# B&R Automation Studio project LAB3FINAL
Automation Studio 

## Configuration Real

### Task classes (Cpu.sw)
```
Cyclic#1 (cycle 2000 us, tolerance 0 us):
  ncsdcctrl <- ncsdcctrl.prg
  SDCAxisCtr <- SDCAxisCtr.prg
DataObjects: Arnc0sys
NcDataObjects: AxisInit <- AxisInit.dob, gAxis03a <- gAxis03obj.gAxis03a.dob, gAxis03i <- gAxis03obj.gAxis03i.dob, AxisApt <- AxisApt.dob, gmcipvar <- GmcIpUserConfig.gmcipvar.dob, gmcipfun <- GmcIpUserConfig.gmcipfun.dob, gmcipfub <- GmcIpUserConfig.gmcipfub.dob, gmcipubr <- GmcIpUserConfig.gmcipubr.dob, gmcipusm <- GmcIpUserConfig.gmcipusm.dob, gmcipui <- GmcIpUserConfig.gmcipui.dob, gmcipus <- GmcIpUserConfig.gmcipus.dob, gmcipuc <- GmcIpUserConfig.gmcipuc.dob, gmcipsys <- GmcIpConfig.gmcipsys.dob, gmciplbr <- GmcIpConfig.gmciplbr.dob, gmcipcbr <- GmcIpConfig.gmcipcbr.dob, gmciplsm <- GmcIpConfig.gmciplsm.dob, gmcipcsm <- GmcIpConfig.gmcipcsm.dob, gmcipcfg <- GmcIpConfig.gmcipcfg.dob, gmcipiec <- GmcIpConfig.gmcipiec.dob, gmciplog <- GmcIpConfig.gmciplog.dob, gmcipesm <- GmcIpConfig.gmcipesm.dob, gmcipmxd <- GmcIpConfig.gmcipmxd.dob, gmcipmx <- GmcIpConfig.gmcipmx.dob, CncInit <- CncInit.dob, CncProg <- CncProg.dob
Binaries: TCData, Acp10map1, acp10cfg, Acp10map, arconfig, User, Role, sysconf, iomap, asfw, ashwd, arnc0cfg, Arnc0map
Libraries: Acp10sdc, Library, Acp10man, Acp10_MC, sys_lib, brsystem, asstring, powerlnk, asieccon, AsMath, Arnc0man, DataObj, AsArLog, FileIO, AsArProf, AsMem, Runtime, astime, Acp10par, NcGlobal, asiotime
```

### Hardware
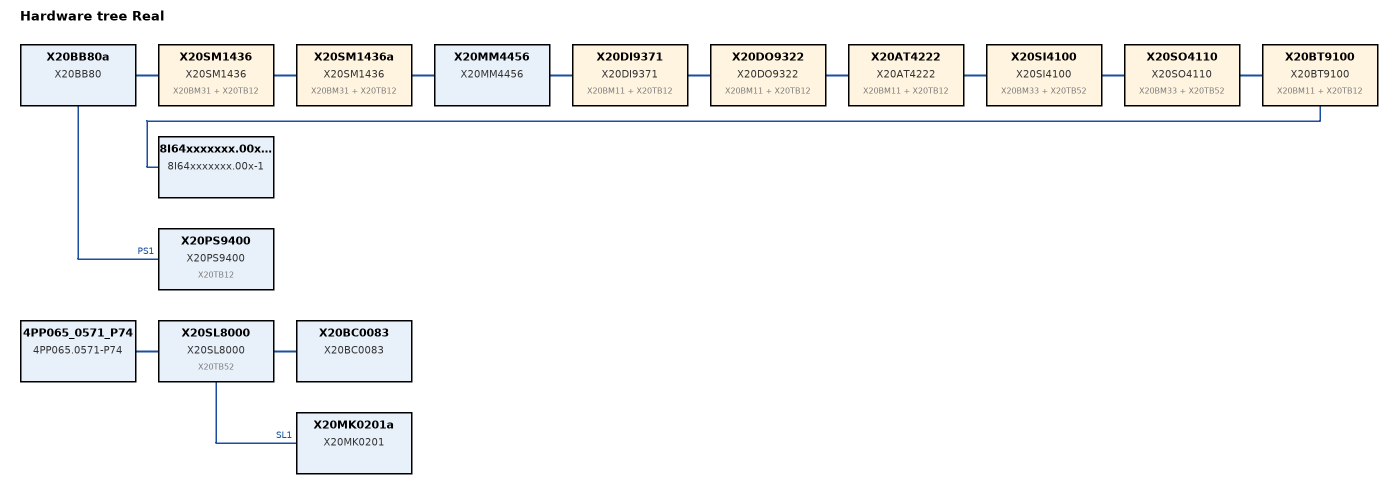
```
4PP065_0571_P74 : 4PP065.0571-P74 v1.1.2.0
  Connector IF4:
    EplInterfaceRedundant = 0
    EplEthInterfaceRedundant = 0
  Connector IF5:
    ActivateDevice = 1
    Mode = Manual
    InternetAddress = 10.0.1.14
    SubnetMask = 255.255.255.0
  ConfigurationID = labBR
  TimerDeviceType = EPLX2X
  TimerDevice = 4PP065_0571_P74.IF4
  TaskClassIdleTime = 2000
  Cyclic1Duration = 2000
  Cyclic1Tolerance = 0
  Cyclic1Output = 1
  Cyclic3Tolerance = 0
  VcObjectName = Visu
8I64xxxxxxx.00x-1 : 8I64xxxxxxx.00x-1 v2.1.2.0  [X2X1 -> X20BT9100.X2X1 [Cable Type=X2XCable, Length=10, Version=1.0.0.2]]
  BothEndSwitchesAreNormallyOpen_r1 = on
  QuickStopIsNormallyOpen_r1 = on
X20AT4222 : X20AT4222 v1.2.3.0  [SS1 -> X20TB12f.SS; SL -> X20BM11c.SL1]
X20BB80a : X20BB80 v1.0.2.0
X20BC0083 : X20BC0083 v2.9.0.0  [PLK1 -> X20SL8000.PLK2 (NodeNumber=2) [Cable Type=PowerlinkCable, Length=10, Version=1.0.0.2]; SL -> X20BB80a.SL1]
X20BM11a : X20BM11 v1.0.0.1  [X2X1 -> X20MM4456.X2X2]
X20BM11b : X20BM11 v1.0.0.1  [X2X1 -> X20BM11a.X2X2]
X20BM11c : X20BM11 v1.0.0.1  [X2X1 -> X20BM11b.X2X2]
X20BM11d : X20BM11 v1.0.0.1  [X2X1 -> X20BM33b.X2X2]
X20BM31a : X20BM31 v1.0.0.1  [X2X1 -> X20BB80a.IF1]
X20BM31b : X20BM31 v1.0.0.1  [X2X1 -> X20BM31a.X2X2]
X20BM33a : X20BM33 v1.0.0.4  [X2X1 -> X20BM11c.X2X2]
X20BM33b : X20BM33 v1.0.0.4  [X2X1 -> X20BM33a.X2X2]
X20BT9100 : X20BT9100 v1.0.3.0  [SS1 -> X20TB12g.SS; SL -> X20BM11d.SL1]
X20DI9371 : X20DI9371 v1.0.2.0  [SS1 -> X20TB12d.SS; SL -> X20BM11a.SL1]
X20DO9322 : X20DO9322 v1.0.3.0  [SS1 -> X20TB12e.SS; SL -> X20BM11b.SL1]
X20MK0201a : X20MK0201 v1.0.0.0  [SL -> X20SL8000.SL1]
X20MM4456 : X20MM4456 v1.4.0.0  [X2X1 -> X20BM31b.X2X2]
X20PS9400 : X20PS9400 v1.0.2.4  [SS1 -> X20TB12b.SS; PS -> X20BB80a.PS1]
X20SI4100 : X20SI4100 v1.10.1.1  [SS1 -> X20TB52b.SS; SL -> X20BM33a.SL1]
X20SL8000 : X20SL8000 v1.6.5.1  [PLK1 -> 4PP065_0571_P74.IF4 (NodeNumber=1) [Cable Type=PowerlinkCable, Length=10, Version=1.0.0.2]; PLK2 -> X20BC0083.PLK1 (NodeNumber=1) [Cable Type=PowerlinkCable, Length=10, Version=1.0.0.2]; SS1 -> X20TB52a.SS]
  SafeProject = SafeLOGIC-1
X20SM1436 : X20SM1436 v1.4.2.1  [SS1 -> X20TB12a.SS; SL -> X20BM31a.SL1]
X20SM1436a : X20SM1436 v1.4.2.1  [SS1 -> X20TB12c.SS; SL -> X20BM31b.SL1]
X20SO4110 : X20SO4110 v1.10.1.1  [SS1 -> X20TB52c.SS; SL -> X20BM33b.SL1]
  SafeLogicID = 2
  SafeModuleID = 3
X20TB12a : X20TB12 v1.0.0.0
X20TB12b : X20TB12 v1.0.0.0
X20TB12c : X20TB12 v1.0.0.0
X20TB12d : X20TB12 v1.0.0.0
X20TB12e : X20TB12 v1.0.0.0
X20TB12f : X20TB12 v1.0.0.0
X20TB12g : X20TB12 v1.0.0.0
X20TB52a : X20TB52 v1.0.0.1
X20TB52b : X20TB52 v1.0.0.1
X20TB52c : X20TB52 v1.0.0.1
```

### IoMap.iom - 4PP065_0571_P74/IoMap.iom
```iecst
VAR_CONFIG
	Cyclic#1.gAxis03_DrvIf.iLifeCnt AT %IB."8I64xxxxxxx.00x-1".SDC_LifeCnt;
	Cyclic#1.gAxis03_DrvIf.iDrvOK AT %IX."8I64xxxxxxx.00x-1".ETAD_Input_Bool_02;
	Cyclic#1.gAxis03_DrvIf.oSetTime AT %QW."8I64xxxxxxx.00x-1".SDC_SetTime;
	Cyclic#1.gAxis03_DrvIf.oSetPos AT %QW."8I64xxxxxxx.00x-1".LFRD_Output;
	Cyclic#1.gAxis03_DiDoIf.iLifeCntDriveReady AT %IB."8I64xxxxxxx.00x-1".SDC_LifeCnt;
	Cyclic#1.gAxis03_DiDoIf.iLifeCntDriveEnable AT %IB."8I64xxxxxxx.00x-1".SDC_LifeCnt;
	Cyclic#1.gAxis03_DiDoIf.oDriveEnable AT %QX."8I64xxxxxxx.00x-1".CMDD_Output_Bool_00;
	Cyclic#1.gAxis03_ModuleOk AT %QX."8I64xxxxxxx.00x-1".CMDD_Output_Bool_01;
	Cyclic#1.gAxis03_ModuleOk AT %QX."8I64xxxxxxx.00x-1".CMDD_Output_Bool_02;
	Cyclic#1.gAxis03_ModuleOk AT %IX."8I64xxxxxxx.00x-1".ModuleOk;
	Cyclic#1.gAxis03_DiDoIf.oDriveEnable AT %QX."8I64xxxxxxx.00x-1".CMDD_Output_Bool_03;
	Cyclic#1.gAxis03_DiDoIf.iDriveReady AT %IX."8I64xxxxxxx.00x-1".ETAD_Input_Bool_02;
	::SDCAxisCtr:pwm_period AT %QW."X20MM4456".PeriodDurationPWM;
	::SDCAxisCtr:axis_X.pwm_value AT %QW."X20MM4456".PulseWidthCurrentPWM01;
	::SDCAxisCtr:axis_X.reset_error AT %QX."X20MM4456".ClearError01;
	::SDCAxisCtr:axis_X.reset_counter AT %QX."X20MM4456".ResetCounter01;
	::SDCAxisCtr:axis_X.counter AT %IW."X20MM4456".Counter01;
	::SDCAxisCtr:axis_X.endswitch_a_reached AT %IX."X20MM4456".StatusInput03; (*Logical condition input 01=Motor 01:A*)
	::SDCAxisCtr:axis_X.endswitch_b_reached AT %IX."X20MM4456".StatusInput04; (*Logical condition input 02=Motor 01:B*)
	::SDCAxisCtr:coil_powered AT %IX."X20DI9371".DigitalInput01;
END_VAR
```

### Acp10map1.ncm - 4PP065_0571_P74/Motion/Acp10map1.ncm
```
NcMapping (NcSwId=ACP10, DisabledNodesAreHidden=False)
  NcObject AxisX (ModuleAddress=SDC_IF1.ST2, InterfaceType=SDC, Type=ncAXIS, Channel=1, AcoposSimulation=Off, InitParameter=AxisInit, AcoposParameter=AxisApt, AdditionalData=CNC_Enabled="1" , Disabled=FALSE, ModuleDisabled=FALSE)
  NcObject AxisY (ModuleAddress=SDC_IF1.ST3, InterfaceType=SDC, Type=ncAXIS, Channel=1, AcoposSimulation=Off, InitParameter=AxisInit, AcoposParameter=AxisApt, AdditionalData=CNC_Enabled="1" , Disabled=FALSE)
  NcObject AxisZ (ModuleAddress=SDC_IF1.ST4, InterfaceType=SDC, Type=ncAXIS, Channel=1, AcoposSimulation=Off, InitParameter=AxisInit, AcoposParameter=AxisApt, AdditionalData=CNC_Enabled="1" , Disabled=FALSE)
```


## Logical view

Binary libraries used (declarations not repeated): Runtime, Operator, AsIecCon, astime, Acp10sdc, Acp10man, Acp10par, NcGlobal, asstring, AsIOTime, Acp10_MC, brsystem, sys_lib, Acp10sim, AsMath, Arnc0man, DataObj, AsArLog, FileIO, AsArProf, AsMem

### Global.var - Global variables
```iecst
VAR
	AxisX : ACP10AXIS_typ := (0);
	AxisX_EncIf : SdcEncIf16_typ := (0);
	AxisX_DrvIf : SdcDrvIf16_typ := (0);
	AxisX_DiDoIf : SdcDiDoIf_typ := (0);
	AxisX_HW : SdcHwCfg_typ := (0);
	gAxisTest : ACP10AXIS_typ := (0);
	gAxisTest_HW : SdcHwCfg_typ := (0);
	gAxisTest_DrvIf : SdcDrvIf16_typ := (0);
	gAxisTest_DiDoIf : SdcDiDoIf_typ := (0);
	gAxisTest_ModuleOk : BOOL := 0;
	gAxis03 : ACP10AXIS_typ := (0);
	gAxis03_HW : SdcHwCfg_typ := (0);
	gAxis03_DrvIf : SdcDrvIf16_typ := (0);
	gAxis03_DiDoIf : SdcDiDoIf_typ := (0);
	gAxis03_ModuleOk : BOOL := 0;
	CNCsys : ARNC0CNC_typ;
END_VAR
```

### Package Logical/Libraries - Global libraries

### Library Logical/Libraries/Library (ANSIC)

#### FB_Axis.c
```c
#include <bur/plctypes.h>
#ifdef __cplusplus
	extern "C"
	{
#endif
	#include "Library.h"
#ifdef __cplusplus
	};
#endif
/* TODO: Add your comment here */
void FB_Axis(struct FB_Axis* inst)
{
	/*
	if (inst->pwm_percentage > 100)
	{
		inst->pwm_percentage = 100;
	}
	if (inst->pwm_percentage < -100)
	{
		inst->pwm_percentage = -100;
	}
	REAL raw_percentage = (REAL) inst->pwm_percentage / 100.0 * 32767.0;
	inst->pwm_value = (INT) raw_percentage;
	*/
	inst->speed = inst->counter - inst->last_counter;
	inst->speed = (inst->speed * 3000 / 24.0) / 0.002;
	inst->last_counter = inst->counter;
}
```

#### FB_Motor.c
```c
#include <bur/plctypes.h>
#ifdef __cplusplus
	extern "C"
	{
#endif
	#include "Library.h"
#ifdef __cplusplus
	};
#endif
/* TODO: Add your comment here */
void FB_Motor(struct FB_Motor* inst)
{
	REAL a = inst->in / inst->k_e - inst->out_w;
	REAL b = a / inst->T_m;
	inst->integrator.dt = inst->dt;
	inst->integrator_phi.dt = inst->dt;
	inst->integrator.in = b;
	FB_Integrator(&inst->integrator);
	inst->out_w = inst->integrator.out;
	inst->integrator_phi.in = inst->out_w;
	FB_Integrator(&inst->integrator_phi);
	inst->out_phi = inst->integrator_phi.out;
}
```

### Package Logical/gAxis03obj - gAxis03obj

### gAxis03i.ax
```
InitParameter (Version=3.13.1, NcSwId=Acp10)
  ACP10AXIS_typ:
    dig_in:
      level:
        reference = ncACTIV_HI
        pos_hw_end = ncACTIV_HI
        neg_hw_end = ncACTIV_HI
        trigger1 = ncACTIV_HI
        trigger2 = ncACTIV_HI
    encoder_if:
      parameter:
        count_dir = ncSTANDARD
        scaling:
          load:
            units = 1000
            rev_motor = 1
    limit:
      parameter:
        v_pos = 10000
        v_neg = 10000
        a1_pos = 50000
        a2_pos = 50000
        a1_neg = 50000
        a2_neg = 50000
        t_jolt = 0
        t_in_pos = 0
        pos_sw_end = 2000000000
        neg_sw_end = -2000000000
        ds_warning = 500
        ds_stop = 1000
        a_stop = 1.0e30
        dv_stop = 0
        dv_stop_mode = ncOFF
    controller:
      mode = ncPOSITION
      position:
        kv = 50
        tn = 0
        t_predict = 0.01
        t_total = 0.01
        p_max = 1.0e30
        i_max = 0
      speed:
        kv = 2.0
        tn = 0
        t_filter = 0.0
        isq_filter1:
          type = ncOFF
          a0 = 0.0
          a1 = 0.0
          b0 = 0.0
          b1 = 0.0
          b2 = 0.0
          c0_par_id = 0
          c1_par_id = 0
        isq_filter2:
          type = ncOFF
          a0 = 0.0
          a1 = 0.0
          b0 = 0.0
          b1 = 0.0
          b2 = 0.0
          c0_par_id = 0
          c1_par_id = 0
        isq_filter3:
          type = ncOFF
          a0 = 0.0
          a1 = 0.0
          b0 = 0.0
          b1 = 0.0
          b2 = 0.0
          c0_par_id = 0
          c1_par_id = 0
      uf:
        type = ncLINEAR
        auto_config = ncMOTOR_PAR
        u0 = 0
        un = 0
        fn = 50.0
        k_f_slip = 0
      ff:
        torque_load = 0.0
        torque_pos = 0.0
        torque_neg = 0.0
        kv_torque = 0.0
        inertia = 0.0
        t_filter_a = 0.0
    move:
      stop:
        parameter[0]:
          decel_ramp = ncA_LIMIT
          controller = ncON
        parameter[1]:
          decel_ramp = ncA_LIMIT
          controller = ncON
        parameter[2]:
          decel_ramp = ncA_LIMIT
          controller = ncON
        parameter[3]:
          decel_ramp = ncA_LIMIT
          controller = ncON
        quickstop:
          decel_ramp = ncA_LIMIT
        drive_error:
          decel_ramp = ncA_LIMIT
      homing:
        parameter:
          s = 0
          v_switch = 5000
          v_trigger = 500
          a = 50000
          mode = ncDIRECT
          edge_sw = ncPOSITIVE
          start_dir = ncPOSITIVE
          trigg_dir = ncPOSITIVE
          ref_pulse = ncOFF
          fix_dir = ncOFF
          tr_s_block = 0
          torque_lim = 0
          ds_block = 0
          ds_stop = 0
      basis:
        parameter:
          v_pos = 5000
          v_neg = 5000
          a1_pos = 50000
          a2_pos = 50000
          a1_neg = 50000
          a2_neg = 50000
    message:
      text:
        parameter:
          format = ncBREAK
          columns = 80
          data_modul = acp10etxen
```

- Data object Logical/GmcIpConfig/gmcipsys (Cnc, version 3.13.0) (no source held here)

### Data object Logical/GmcIpConfig/gmciplbr (Cnc)

#### gmciplbr.cnc
```
Root (LangModule=ailgcode, Version=1.0)
  BuiltInProcs:
    cancel = beginpathsynch
        StopCyclicGroups(:${*}:);
      endpathsynch (MinArgs=1, MaxArgs=*)
  BuiltInFns (PatternSuffix=:\[)
    ABS = Abs(:$[1]:) (NumArgs=1, Inline=Yes)
    SQR = ($[1] * $[1]) (NumArgs=1)
    ACOS = ACos(:$[1]:) (NumArgs=1, Inline=Yes)
    ASIN = ASin(:$[1]:) (NumArgs=1, Inline=Yes)
    ATAN = ATan(:$[1]:) (NumArgs=1, Inline=Yes)
    COS = Cos(:$[1]:) (NumArgs=1, Inline=Yes)
    DEXP = DExp(:$[1]:) (NumArgs=1, Inline=Yes)
    EXP = Exp(:$[1]:) (NumArgs=1, Inline=Yes)
    FIX = Fix(:$[1]:) (NumArgs=1, Inline=Yes)
    FRACT = Fract(:$[1]:) (NumArgs=1, Inline=Yes)
    FUP = Fup(:$[1]:) (NumArgs=1, Inline=Yes)
    INV = ~($[1]) (NumArgs=1, Inline=Yes)
    LN = Ln(:$[1]:) (NumArgs=1, Inline=Yes)
    LOG = Log(:$[1]:) (NumArgs=1, Inline=Yes)
    ROUND = ToInt(:$[1]:) (NumArgs=1, Inline=Yes)
    SIN = Sin(:$[1]:) (NumArgs=1, Inline=Yes)
    SQRT = Sqrt(:$[1]:) (NumArgs=1, Inline=Yes)
    TAN = Tan(:$[1]:) (NumArgs=1, Inline=Yes)
    BOOL = ToBool(:$[1]:) (NumArgs=1, Inline=Yes)
    INT = Fix(:$[1]:) (NumArgs=1, Inline=Yes)
    ADR = Adr(:\$[1]:) (NumArgs=1, Inline=Yes)
    SIZEOF = Sizeof(:\$[1]:) (NumArgs=1, Inline=Yes)
    NUM_LOADED_FILES = NumLoadedFiles(::) (NumArgs=0)
    NUM_LOADED_PROG_FILES = NumLoadedProgFiles(::) (NumArgs=0)
    MEM_SIZE_IP_ALL = MemSizeIpInstAll(::) (NumArgs=0)
    MEM_SIZE_IP_LIB = MemSizeIpInst(::) (NumArgs=0)
    MEM_SIZE_SHLIB = MemSizeShLib(::) (NumArgs=0)
    MEM_SIZE_FILE = MemSizeFile(:$[1]:) (MinArgs=0, MaxArgs=1)
    MEM_SIZE_IP_STACK_SPACE = MemStackSpace(::) (NumArgs=0)
  AxesSpec:
    AxisRef = $\s*=\s*AC (Mode=3)
    AxisRef = $\s*=\s*IC (Mode=4)
  PVMacros:
    RDISABLE (ArrayDims=0, Group=500)
      CALL = @#job->sa.keep_alive = 1;
        @#thread.sa_keep_alive = 1; (Inline=Yes)
  Parameters:
    R (IndexType=RParamIndex, ValueType=FLOAT)
      ARG (ref=EXPR, DataType=RParamIndex)
    P (IndexType=RParamIndex, ValueType=FLOAT)
      ARG (ref=EXPR, DataType=RParamIndex)
    EXB (IndexType=EXParamIndex, ValueType=Byte)
      ARG (ref=EXPR, DataType=EXParamIndex)
    EXW (IndexType=EXParamIndex, ValueType=Word)
      ARG (ref=EXPR, DataType=EXParamIndex)
    EXL (IndexType=EXParamIndex, ValueType=Long)
      ARG (ref=EXPR, DataType=EXParamIndex)
    EXF (IndexType=EXFParamIndex, ValueType=FLOAT)
      ARG (ref=EXPR, DataType=EXFParamIndex)
    MW (Synchronous=Yes, IndexType=MParamIndex, ValueType=Word)
      ARG (ref=EXPR, DataType=MParamIndex)
    ML (Synchronous=Yes, IndexType=MParamIndex, ValueType=Long)
      ARG (ref=EXPR, DataType=MParamIndex)
    MF (Synchronous=Yes, IndexType=MParamIndex, ValueType=FLOAT)
      ARG (ref=EXPR, DataType=MParamIndex)
  PrimTypes (PatternSuffix=:[^\[], MapIECTypes=Yes)
  Preprocess:
    PP_RULE_FRAME_I (Search=$FRAME_I, Replace=[1,0,0,0,1,0,0,0,1,0,0,0])
    PP_RULE_FRAME_DEF (IsPattern=Yes, Search=FRAME:[^\w\d], Replace=LREAL{12})
  FubTemplates:
    StdFubTemplate (IsDefault=Yes, Inline=Yes)
      Arg (ref=FUBINST, DataType=FLOAT)
      Arg (ref=FUBERRLEV, DataType=FLOAT)
      Arg (ref=PATHSYNCH, DataType=FLOAT)
      Arg (ref=BLOCKING, DataType=FLOAT)
  SynchActions:
    SABlocks:
      default (IsDefault=Yes)
        cyclic (Inline=Yes)
          Arg (ref=ACTIONS, DataType=STATEMENTS)
          Arg (ref=ID, DataType=FLOAT, DefaultInt=-1, MinCount=0, MaxCount=1)
      whenever:
        cyclic (Inline=Yes)
          Arg (ref=COND, DataType=FLOAT)
          Arg (ref=ACTIONS, DataType=STATEMENTS)
          Arg (ref=ID, DataType=FLOAT, DefaultInt=-1, MinCount=0, MaxCount=1)
      when:
        cyclic (Inline=Yes)
          Arg (ref=COND, DataType=FLOAT)
          Arg (ref=ACTIONS, DataType=STATEMENTS)
          Arg (ref=ID, DataType=FLOAT, DefaultInt=-1, MinCount=0, MaxCount=1)
      every:
        cyclic (Inline=Yes)
          Arg (ref=COND, DataType=FLOAT)
          Arg (ref=ACTIONS, DataType=STATEMENTS)
          Arg (ref=ID, DataType=FLOAT, DefaultInt=-1, MinCount=0, MaxCount=1)
      from:
        cyclic (Inline=Yes)
          Arg (ref=COND, DataType=FLOAT)
          Arg (ref=ACTIONS, DataType=STATEMENTS)
          Arg (ref=ID, DataType=FLOAT, DefaultInt=-1, MinCount=0, MaxCount=1)
    NonModalActivation:
      Start = @#thread.sa_last_keep_alive = 1;
        ActivateCyclicGroup(:-1:);
      Stop = WaitStopCyclicGroups(:(:-1:):);
  ParserData (NestedComments=Yes, DefaultCaseSensitive=No, CommentsSpanLines=No, SubDeclsLocalToFile=Yes, ProgDeclsLocalToFile=Yes, AllowUnprefixedFileCalls=No, LocalVarScopeForMainProg=No, FileScopeVarsVisibleInSub=Yes, MainPrgReturnAtNextMainPrgHdr=Yes, MaxSizePassByValue=1024, AllowVarReadBeforeAssign=No, AllowArrayRefWithoutIndex=Yes, AllowStructMemberAutoDereference=Yes, AllowVariableAutoDereference=Yes, AllowIgnoredExtraSubArgs=Yes, EnableStringCharacterIndexing=Yes, OnMacroRedefinition=Warn, CheckFileTimestampBeforeCalls=Yes)
    TKG_END_OF_LINE = \n (IsPattern=No)
    TKG_LINE_CONTINUE = \ (IsPattern=No, FileXLInvalid=Yes)
    TKG_LINE_BREAK = @@
    TKG_ARITH_BINARY_MODULO = MOD
    TKG_TRUE = TRUE:\W (IsPattern=Yes)
    TKG_FALSE = FALSE:\W (IsPattern=Yes)
    TKG_PAREVAL_MODAL_ID = ID:[\s=] (FileXLInvalid=Yes, IsPattern=Yes)
    TKG_OPEN_COMMENT = (
    TKG_CLOSE_COMMENT = )
    TKG_OPEN_BRACKET = [
    TKG_COMMA = ,
    TKG_CLOSE_BRACKET = ]
    TKG_OPEN_INDEXBRACKET = {
    TKG_CLOSE_INDEXBRACKET = }
    TKG_NUMBER = \d+\.\d+|\d+\.:[^\.] (IsPattern=Yes)
    TKG_INTEGER = \d+ (IsPattern=Yes)
    TKG_FRACTION = \.\d+ (IsPattern=Yes)
    TKG_DOT = \.:\w (IsPattern=Yes, FollowedBy=TKG_STRUCT_MEMBER_REF)
    TKG_STRUCT_MEMBER_REF = \w|\w[\w\d]+ (IsPattern=Yes, Restricted=Yes)
    TKG_NUMBER_EXP = EX:[\s\d\+\-\.] (IsPattern=Yes)
    TKG_MACRO_DEFINE_GLOBAL = define\s+ip_global:\s (IsPattern=Yes, FollowedBy=TKG_MACRO_NAME)
    TKG_MACRO_DEFINE = define\s+local:\s|define:\s (IsPattern=Yes, FollowedBy=TKG_MACRO_NAME)
    TKG_MACRO_UNDEFINE = undefine:\s (IsPattern=Yes, FollowedBy=TKG_MACRO_NAME)
    TKG_MACRO_AS = as:[\s\n] (IsPattern=Yes, FollowedBy=TKG_MACRO_TEXT)
    TKG_MACRO_NAME = [$\w][$\w\d]+ (Restricted=Yes, IsPattern=Yes)
    TKG_MACRO_TEXT = . (Restricted=Yes, IsPattern=Yes)
    TKG_BUILTIN_NUM_FN_NAME
    _TKG_LABEL_DEF1:
      TKG_LABEL_DEF = L[\w\d]+:\:[^\w\d] (IsPattern=Yes, FollowedBy=TKG_LABEL_SUFFIX)
    TKG_SUBPROG_START = %:L (FileXLInvalid=Yes, IsPattern=Yes, FollowedBy=TKG_SUBPROG_NAME)
    TKG_SUBPROG_NAME = L\d+ (IsPattern=Yes, Restricted=Yes)
    TKG_SUBPROG_CALL = L:L\d (IsPattern=Yes, FollowedBy=TKG_SUBPROG_NAME)
    TKG_SUBPROG_PROTO = %D:L (IsPattern=Yes, FollowedBy=TKG_SUBPROG_NAME)
    TKG_SUBCALL_REPEAT_PREFIX = O:[\s\d] (IsPattern=Yes, FollowedBy=TKG_INTEGER)
    TKG_EXTERN = EXTERN:\s (IsPattern=Yes, FollowedBy=TKG_PROG_FILE_NAME)
    TKG_ARG_PASSBYREF = VAR\s (IsPattern=Yes)
    TKG_SET_MODAL_SUB = MCALL:\W (FileXLInvalid=Yes, IsPattern=Yes)
    TKG_PROG_START = %:\d (IsPattern=Yes, FollowedBy=TKG_PROG_NAME)
    TKG_PROG_NAME = \d+ (IsPattern=Yes, Restricted=Yes)
    TKG_PROG_CALL = L:[^L] (IsPattern=Yes, FollowedBy=TKG_PROG_FILE_NAME)
    TKG_PROG_FILE_NAME = [\^#&@']?[\w\d\.\\]+:[^\w\d\.\\\:]|[\^#][\w\d]+\:[\w\d\.\\]+ (IsPattern=Yes, Restricted=Yes)
    TKG_SUPPRESS_SINGLE_STEP = NOHALT
    TKG_NC_BLOCK_PREFIX = N:[\d\s] (IsPattern=Yes)
    TKG_PARAM_PREFIX = R:\d|P:\d|M[WLF]:\d|EX[WLBF]:\d (IsPattern=Yes)
    TKG_SUBRANGE = ..
    TKG_G_CODE_PREFIX = G:[\s\d] (IsPattern=Yes)
    TKG_M_CODE_PREFIX = M:[\s\d\[] (IsPattern=Yes)
    TKG_PAREVAL_DO = do:\s (FileXLInvalid=Yes, IsPattern=Yes)
    TKG_GOTO = $GOTO:\s (FileXLInvalid=Yes, IsPattern=Yes, OptFollowedBy=TKG_GOTO_DEST)
    TKG_GOTO_DEST = \w[\w\d]* (IsPattern=Yes, Restricted=Yes)
    TKG_LOGICAL_BINARY_AND = &&
    TKG_LOGICAL_BINARY_OR = ||
    TKG_LOGICAL_BINARY_XOR = XOR
    TKG_STRING_CONCAT = <<
    TKG_COMP_BINARY_GREATER_THAN_OR_EQ = >=
    TKG_COMP_BINARY_LESS_THAN_OR_EQ = <=
    TKG_COMP_BINARY_EQUAL_TO = ==
    TKG_COMP_BINARY_NOT_EQUAL_TO = !=
    TKG_COMP_BINARY_GREATER_THAN = >
    TKG_COMP_BINARY_LESS_THAN = <
    TKG_ASSIGN_EQ = =
    TKG_LOGICAL_UNARY_NOT = !
    TKG_BITWISE_BINARY_AND = &
    TKG_BITWISE_BINARY_OR = |
    TKG_BITWISE_BINARY_XOR = ^
    TKG_BITWISE_UNARY_COMPLEMENT = ~
    TKG_ARITH_BINARY_PLUS = +
    TKG_ARITH_BINARY_MINUS = -
    TKG_ARITH_BINARY_POWER = **
    TKG_ARITH_BINARY_MULTIPLY = *
    TKG_ARITH_BINARY_DIVIDE = /
    TKG_IF = $IF (FileXLInvalid=Yes)
    TKG_THEN = $THEN (FileXLInvalid=Yes)
    TKG_BLOCK_ELSEIF = $ELSEIF (FileXLInvalid=Yes)
    TKG_BLOCK_ELSE = $ELSE (FileXLInvalid=Yes)
    TKG_BLOCK_ENDIF = $ENDIF (FileXLInvalid=Yes)
    TKG_SWITCH = $SWITCH (FileXLInvalid=Yes)
    TKG_SWITCH_CASE = $CASE (FileXLInvalid=Yes)
    TKG_SWITCH_DEFAULT = $DEFAULT (FileXLInvalid=Yes)
    TKG_ENDSWITCH = $ENDSWITCH (FileXLInvalid=Yes)
    TKG_FOR = $FOR (FileXLInvalid=Yes)
    TKG_ENDFOR = $ENDFOR (FileXLInvalid=Yes)
    TKG_WHILE = $WHILE (FileXLInvalid=Yes)
    TKG_ENDWHILE = $ENDWHILE (FileXLInvalid=Yes)
    TKG_DO = $DO (FileXLInvalid=Yes)
    TKG_ENDDO = $ENDDO (FileXLInvalid=Yes)
    TKG_BREAK = $BREAK (FileXLInvalid=Yes)
    TKG_CONTINUE = $CONTINUE (FileXLInvalid=Yes)
    TKG_PRIM_TYPE (IsPattern=Yes)
    TKG_PV_DECL = def:\s (IsPattern=Yes)
    TKG_PV_UNDECL = ~def:\s (IsPattern=Yes)
    TKG_PV_DECL_REF = \w[\w\d\.\:\*]+|\w (IsPattern=Yes, Restricted=Yes)
    TKG_VARSCOPE_IP_LOCAL = local:[\s\n] (IsPattern=Yes)
    TKG_VARSCOPE_IP_GLOBAL = ip_global:[\s\n] (IsPattern=Yes)
    TKG_VARSCOPE_NC_GLOBAL = nc_global:[\s\n] (IsPattern=Yes)
    TKG_VARSCOPE_PLC_GLOBAL = plc_global:[\s\n] (IsPattern=Yes)
    TKG_VAR_RETAIN = retain:\s (IsPattern=Yes)
    TKG_VARSYNCH_IP = ip_synch:\s (IsPattern=Yes)
    TKG_VARSYNCH_PATH = path_synch:\s (IsPattern=Yes)
    TKG_LABEL_DEF = \w:\:|\w[\w\d]+:\: (IsPattern=Yes, FollowedBy=TKG_LABEL_SUFFIX)
    TKG_LABEL_SUFFIX = : (Restricted=Yes)
    TKG_FUB_DECL = fub:\s (IsPattern=Yes)
    TKG_FUB_ERR_LEV_1 = error_level_1:\s (IsPattern=Yes)
    TKG_FUB_ERR_LEV_2 = error_level_2:\s (IsPattern=Yes)
    TKG_FUB_ERR_LEV_3 = error_level_3:\s (IsPattern=Yes)
    TKG_FUB_ERR_LEV_4 = error_level_4:\s (IsPattern=Yes)
    TKG_FUB_BLOCKING = blocking:\s (IsPattern=Yes)
    TKG_FUB_NON_BLOCKING = non_blocking:\s (IsPattern=Yes)
    TKG_IEC_TYPED_VALUE = #[\w\d]+ (IsPattern=Yes)
    TKG_REFERENCE = ref:[\s\n]|reference:[\s\n] (IsPattern=Yes, FollowedBy=TKG_IEC_TO)
    TKG_IEC_TO = to:[\s\n] (IsPattern=Yes, Restricted=Yes)
    TKG_ACCESS = ACCESS:[\s\n] (IsPattern=Yes)
    TKG_WORD = \w|\w[\w\d\.]+ (IsPattern=Yes)
  StringChars (AsciiStringStart=", UTF16StringStart=W", UTF16StringEnd=")
    EscapeSeq (Search=$N, ReplaceValue=10)
    EscapeSeq (Search=$L, ReplaceValue=10)
    EscapeSeq (Search=$P, ReplaceValue=12)
    EscapeSeq (Search=$R, ReplaceValue=13)
    EscapeSeq (Search=$T, ReplaceValue=9)
    EscapeSeq (Search=$Q, ReplaceStr=")
    EscapeSeq (Search=$', ReplaceStr=')
    EscapeSeq (Search=$", ReplaceStr=")
    EscapeSeq (Search=$[\dA-Fa-f]+, IsPattern=Yes, ReplaceEncodingBase=16)
    EscapeSeq (Search=$$, ReplaceStr=$)
    EscapeSeq (Search=$, ReplaceStr=)
```

- Data object Logical/GmcIpConfig/gmcipcbr (Cnc, version 3.13.0) (no source held here)

### Data object Logical/GmcIpConfig/gmcipcsm (Cnc)

#### gmcipcsm.cnc
```
Root (LangModule=ailgcode, Version=1.0)
  Constants:
    NumAxes = 15 (Type=INT)
  Preprocess:
    PP_RULE_STOPRE (Search=STOPRE, Replace=G172)
    PP_RULE_CIP (Search=CIP:\W, Replace=G102, IsPattern=Yes)
  Types:
    RotationAngleSpecifier (type=ENUM, EnumType=REGEXP, Value6=H)
    RadiusSpecifier (type=ENUM, EnumType=REGEXP, Value1=R\s*=, Value2=CR\s*=)
    InterpolParam (type=ENUM, EnumType=REGEXP, Value0=I, Value1=J, Value2=K, Value100=G161\s*I, Value101=G161\s*J, Value102=G161\s*K, Value200=G162\s*I, Value201=G162\s*J, Value202=G162\s*K, Value0300=I\s*=\s*AC, Value0301=J\s*=\s*AC, Value0302=K\s*=\s*AC, Value0400=I\s*=\s*IC, Value0401=J\s*=\s*IC, Value0402=K\s*=\s*IC)
    CirclePointParam (type=ENUM, EnumType=REGEXP, Value0=I1\s*=, Value1=J1\s*=, Value2=K1\s*=, Value100=G161\s*I1\s*=, Value101=G161\s*J1\s*=, Value102=G161\s*K1\s*=, Value200=G162\s*I1\s*=, Value201=G162\s*J1\s*=, Value202=G162\s*K1\s*=, Value0300=I1\s*=\s*AC, Value0301=J1\s*=\s*AC, Value0302=K1\s*=\s*AC, Value0400=I1\s*=\s*IC, Value0401=J1\s*=\s*IC, Value0402=K1\s*=\s*IC)
    RPYAngleName (type=ENUM, EnumType=REGEXP, Value1=ROLL, Value0=PITCH, Value2=YAW)
    EulerAngleName (type=ENUM, EnumType=REGEXP, Value3=PHI, Value4=THETA, Value5=PSI)
    RotaryVectorName (type=ENUM, EnumType=REGEXP, Value0=P\s*=, Value1=Q\s*=, Value2=R\s*=)
    DwellTime (type=FLOAT)
    RParamIndex (type=INT, MinValue=0, MaxValue=999)
    EXParamIndex (type=INT, MinValue=0, MaxValue=99)
    MParamIndex (type=INT, MinValue=0, MaxValue=99)
    Byte (type=INT, MinValue=0, MaxValue=255)
    Word (type=INT, MinValue=-32768, MaxValue=32767)
    Long (type=INT)
  PVMacros:
    SAVE (ArrayDims=0, Group=500)
      CALL = Info(:id:52101, msg:"Save Modal GCode State NOT SUPPORTED YET":);
  SysVars
  Parameters:
    R (IndexType=RParamIndex, ValueType=FLOAT)
      ARG (ref=EXPR, DataType=RParamIndex)
    QUOTED (QuotedName=$R, Synchronous=Yes, IndexType=RParamIndex, ValueType=FLOAT)
      ARG (ref=EXPR, DataType=RParamIndex)
    QUOTED (QuotedName=$P, Synchronous=Yes, IndexType=RParamIndex, ValueType=FLOAT)
      ARG (ref=EXPR, DataType=RParamIndex)
    EXB (IndexType=EXParamIndex, ValueType=Byte)
      ARG (ref=EXPR, DataType=EXParamIndex)
    EXW (IndexType=EXParamIndex, ValueType=Word)
      ARG (ref=EXPR, DataType=EXParamIndex)
    EXL (IndexType=EXParamIndex, ValueType=Long)
      ARG (ref=EXPR, DataType=EXParamIndex)
    EXF (IndexType=EXFParamIndex, ValueType=FLOAT)
      ARG (ref=EXPR, DataType=EXFParamIndex)
    MW (Synchronous=Yes, IndexType=MParamIndex, ValueType=Word)
      ARG (ref=EXPR, DataType=MParamIndex)
    ML (Synchronous=Yes, IndexType=MParamIndex, ValueType=Long)
      ARG (ref=EXPR, DataType=MParamIndex)
    MF (Synchronous=Yes, IndexType=MParamIndex, ValueType=FLOAT)
      ARG (ref=EXPR, DataType=MParamIndex)
  MCodes:
    M17 = 17 (Group=41, Alias=RET:[^\d\w\(], Eval=Early, Inline=Yes, AliasIsPattern=Yes)
      ARG (ref=VALUE, DataType=FLOAT, RequireLiteral=Yes)
    M17_1 = 17.1 (Group=41, Alias=CONDRET, Eval=Early, Inline=Yes)
      ARG (ref=VALUE, DataType=FLOAT, RequireLiteral=Yes)
```

### Data object Logical/GmcIpConfig/gmciplog (Cnc)

#### gmciplog.cnc
```
Root (LangModule=ailgcode, Version=1.0)
  AxesSpec
  PVMacros:
    DR8:
      REF = #next_motion.Data.R8_value
    DI4:
      REF = #next_motion.Data.I4_value
    DU4:
      REF = #next_motion.Data.UI4_value
    DR8_G211:
      SET = %_CNC.TA = ${EXPR};
       if (%_CNC.TA < 0)
         %_CNC.TA = 0;
       endif
        #next_motion.Data.R8_value = ${EXPR};
    Dlp:
      REF = #next_motion.Data.LinMovement.Position
    Dli:
      SET = #next_motion.Data.LinMovement.Idx[0] = ArrayRep(:(:-1:):);
        #next_motion.Data.LinMovement.Idx = ${EXPR};
    Dlm:
      SET = #next_motion.Data.LinMovement.Mode[0] = ArrayRep(:(:-1:):);
        #next_motion.Data.LinMovement.Mode = ${EXPR};
    Dto:
      REF = #next_motion.Data.Trans.Offset
    Dti:
      SET = #next_motion.Data.Trans.AxIdx[0] = ArrayRep(:(:-1:):);
        #next_motion.Data.Trans.AxIdx = ${EXPR};
    Dtm:
      SET = #next_motion.Data.Trans.Mode[0] = ArrayRep(:(:-1:):);
        #next_motion.Data.Trans.Mode = ${EXPR};
    DSPp:
      REF = #next_motion.Data.SplinePoint.Position
    DSPi:
      SET = #next_motion.Data.SplinePoint.AxIdx[0] = ArrayRep(:(:-1:):);
        #next_motion.Data.SplinePoint.AxIdx = ${EXPR};
    DSPm:
      SET = #next_motion.Data.SplinePoint.Mode[0] = ArrayRep(:(:-1:):);
        #next_motion.Data.SplinePoint.Mode = ${EXPR};
    Dcp:
      REF = #next_motion.Data.CircMovement.Parameter
    Dci:
      SET = #next_motion.Data.CircMovement.Idx[0] = ArrayRep(:(:-1:):);
        #next_motion.Data.CircMovement.Idx = ${EXPR};
    Dcm:
      SET = #next_motion.Data.CircMovement.Mode[0] = ArrayRep(:(:-1:):);
        #next_motion.Data.CircMovement.Mode = ${EXPR};
    Dtp:
      REF = #next_motion.Data.ToolAxOrient.Parameter
    Dts:
      REF = #next_motion.Data.ToolAxOrient.Sign
    Daz:
      REF = #next_motion.Data.AbsZeroPtShift.ZpRecIdx
    Dpt:
      SET = #next_motion.Data.ProgZeroPtShift.Type[0] = ArrayRep(:(:-1:):);
        #next_motion.Data.ProgZeroPtShift.Type = ${EXPR};
    Dpm:
      SET = #next_motion.Data.ProgZeroPtShift.Mode[0] = ArrayRep(:(:-1:):);
        #next_motion.Data.ProgZeroPtShift.Mode = ${EXPR};
    Dpa:
      REF = #next_motion.Data.ProgZeroPtShift.AxShift
    Dovpathdef:
      REF = #next_motion.Data.OptMotPar.path_definition
    Dovpathdefd:
      REF = #next_motion.Data.OptMotPar.path_definition_def
    Dorpar:
      REF = #next_motion.Data.OptMotPar.robot_par
    Dorpard:
      REF = #next_motion.Data.OptMotPar.robot_par_def
    Dolim:
      REF = #next_motion.Data.OptMotPar.limits_idx
    Dolimd:
      REF = #next_motion.Data.OptMotPar.limits_idx_def
    Dolimfac:
      REF = #next_motion.Data.OptMotPar.limits_factor
    Dolimfacd:
      REF = #next_motion.Data.OptMotPar.limits_factor_def
    Dfdx:
      REF = #next_motion.Data.FullTrfTool.Dx
    Dfdy:
      REF = #next_motion.Data.FullTrfTool.Dy
    Dfdz:
      REF = #next_motion.Data.FullTrfTool.Dz
    Dfph:
      REF = #next_motion.Data.FullTrfTool.Phi
    Dft:
      REF = #next_motion.Data.FullTrfTool.Theta
    Dfps:
      REF = #next_motion.Data.FullTrfTool.Psi
    DPLDli:
      REF = #next_motion.Data.PosLatchDistance.LatchIdx
    DPLDts:
      REF = #next_motion.Data.PosLatchDistance.TriggSource
    DPLDe:
      REF = #next_motion.Data.PosLatchDistance.Edge
    DPLDti:
      REF = #next_motion.Data.PosLatchDistance.HwTrigIdx
    DPLDd:
      REF = #next_motion.Data.PosLatchDistance.Distance
    DPLli:
      REF = #next_motion.Data.PosLatch.LatchIdx
    DPLts:
      REF = #next_motion.Data.PosLatch.TriggSource
    DPLe:
      REF = #next_motion.Data.PosLatch.Edge
    DPLti:
      REF = #next_motion.Data.PosLatch.HwTrigIdx
    Drma:
      REF = #next_motion.Data.R_DependFeed.MaxRadius
    Drmi:
      REF = #next_motion.Data.R_DependFeed.MinRadius
    Drr:
      REF = #next_motion.Data.R_DependFeed.Rate
    Dsvp:
      SET = #next_motion.Data.Set_v_jump.programmed[0] = ArrayRep(:(:ncOFF:):);
        #next_motion.Data.Set_v_jump.programmed = ${EXPR};
    Dsvv:
      REF = #next_motion.Data.Set_v_jump.value
    Dsap:
      SET = #next_motion.Data.Set_a_jump.programmed[0] = ArrayRep(:(:ncOFF:):);
        #next_motion.Data.Set_a_jump.programmed = ${EXPR};
    Dsav:
      REF = #next_motion.Data.Set_a_jump.value
    Dsep:
      SET = #next_motion.Data.SetAxLimit.programmed[0] = ArrayRep(:(:ncOFF:):);
        #next_motion.Data.SetAxLimit.programmed = ${EXPR};
    Dser:
      REF = #next_motion.Data.SetAxLimit.RecordIdx
    Dcad:
      REF = #next_motion.Data.CamWrapping.Diameter
    Dcap:
      REF = #next_motion.Data.CamWrapping.ParameterP1
    Dsu:
      REF = #next_motion.Data.SetPathAccDec.UnitType
    Dsv108:
      SET = #next_motion.Data.SetPathAccDec.value = ${EXPR};
        if (#next_motion.Data.SetPathAccDec.UnitType == 1)
          %_CNC.lim_path_acc_p = ${EXPR} / 100.0 * %_CNC.lim_path_acc_p_ini;
        else
          %_CNC.lim_path_acc_p = ${EXPR};
        endif
    Dsv109:
      SET = #next_motion.Data.SetPathAccDec.value = ${EXPR};
        if (#next_motion.Data.SetPathAccDec.UnitType == 1)
          %_CNC.lim_path_acc_n = ${EXPR} / 100.0 * %_CNC.lim_path_acc_n_ini;
        else
          %_CNC.lim_path_acc_n = ${EXPR};
        endif
    Dsv110:
      SET = #next_motion.Data.SetPathAccDec.value = ${EXPR};
        if (#next_motion.Data.SetPathAccDec.UnitType == 1)
          %_CNC.lim_path_acc_p = ${EXPR} / 100.0 * %_CNC.lim_path_acc_p_ini;
          %_CNC.lim_path_acc_n = ${EXPR} / 100.0 * %_CNC.lim_path_acc_n_ini;
        else
          %_CNC.lim_path_acc_p = ${EXPR};
          %_CNC.lim_path_acc_n = ${EXPR};
        endif
    Dsma:
      REF = #next_motion.Data.SetTransSpeed.MaxAngle
    Dsmi:
      REF = #next_motion.Data.SetTransSpeed.MinAngle
    Dsr:
      REF = #next_motion.Data.SetTransSpeed.RedFactor
    Dbrp:
      REF = #next_motion.Data.BezierSpline.RadiusProgrammed
    Dbr:
      REF = #next_motion.Data.BezierSpline.Radius
    Dbvp:
      REF = #next_motion.Data.BezierSpline.VeProgrammed
    Dbv:
      REF = #next_motion.Data.BezierSpline.Ve
    Dbl:
      REF = #next_motion.Data.BezierSpline.LinProgrammed
    Dbsf:
      REF = #next_motion.Data.BezierSpline.scalingFactor
    Dbsfd:
      REF = #next_motion.Data.BezierSpline.scalingFactor_def
    Dao:
      REF = #next_motion.Data.AutomTangentialAx.Offset
    Daa:
      REF = #next_motion.Data.AutomTangentialAx.AxIdx
    DAMa:
      REF = #next_motion.Data.AxisMapping.AxIdx
    DAMf:
      REF = #next_motion.Data.AxisMapping.factor
    DAMp:
      REF = #next_motion.Data.AxisMapping.ParameterP1
    DSPEt:
      REF = #next_motion.Data.SignalPathEnd.Time
    DSPEst:
      REF = #next_motion.Data.SignalPathEnd.SignalType
    DSPEsi:
      REF = #next_motion.Data.SignalPathEnd.SignalIdx
    DSPEsd:
      REF = #next_motion.Data.SignalPathEnd.SourceData
    DSPEd:
      REF = #next_motion.Data.SignalPathEnd.DataLength
    DSPEp:
      SET = #next_motion.Data.SignalPathEnd.pDestination = \#sys_vars.EXF[0];
    DSPEDst:
      REF = #next_motion.Data.SignalPathEndDist.SignalType
    DSPEDsi:
      REF = #next_motion.Data.SignalPathEndDist.SignalIdx
    DSPEDsd:
      REF = #next_motion.Data.SignalPathEndDist.SourceData
    DSPEDd:
      REF = #next_motion.Data.SignalPathEndDist.DataLength
    DSPEDp:
      SET = #next_motion.Data.SignalPathEndDist.pDestination = \#sys_vars.EXF[0];
    DSPo:
      REF = #next_motion.Data.SignalPredict.Override
    DWCx1:
      REF = #next_motion.Data.WS_Ctrl.x1
    DWCz1:
      REF = #next_motion.Data.WS_Ctrl.z1
    DWCy1:
      REF = #next_motion.Data.WS_Ctrl.y1
    DWCx2:
      REF = #next_motion.Data.WS_Ctrl.x2
    DWCz2:
      REF = #next_motion.Data.WS_Ctrl.y2
    DWCy2:
      REF = #next_motion.Data.WS_Ctrl.z2
    DWCi:
      REF = #next_motion.Data.WS_Ctrl.index
    DWCc:
      REF = #next_motion.Data.WS_Ctrl.coord
    DWCp:
      REF = #next_motion.Data.WS_Ctrl.pplane
    DWCo:
      REF = #next_motion.Data.WS_Ctrl.orient
    DWCs:
      REF = #next_motion.Data.WS_Ctrl.shape
    DWCa:
      SET = #next_motion.Data.WS_Ctrl.arm_diameter[0] = ArrayRep(:(:ncOFF:):);
        #next_motion.Data.WS_Ctrl.arm_diameter = ${EXPR};
    DTDRt:
      REF = #next_motion.Data.ToolDataRecord.ToolIdx
    Sz:
      REF = #sys_vars.ZP
    DSSi:
      REF = #next_motion.Data.SpindleSpeed.Idx
    DSSs:
      REF = #next_motion.Data.SpindleSpeed.speed
    DCSSt:
      REF = #next_motion.Data.C2_SplineStart.BCType
    DCSSv:
      REF = #next_motion.Data.C2_SplineStart.BCValue
    DCSSp:
      SET = #next_motion.Data.C2_SplineStart.BCProgrammed[0] = ArrayRep(:(:ncOFF:):);
        #next_motion.Data.C2_SplineStart.BCProgrammed = ${EXPR};
    DCSSsp:
      REF = #next_motion.Data.C2_SplineStart.SegmentParameter
    DCSSst:
      REF = #next_motion.Data.C2_SplineStart.SegmentType
    DCSEt:
      REF = #next_motion.Data.C2_SplineEnd.BCType
    DCSEv:
      REF = #next_motion.Data.C2_SplineEnd.BCValue
    DCSEp:
      SET = #next_motion.Data.C2_SplineEnd.BCProgrammed[0] = ArrayRep(:(:ncOFF:):);
        #next_motion.Data.C2_SplineEnd.BCProgrammed = ${EXPR};
    DFd:
      REF = #next_motion.Data.Frame.Data
    DSVs:
      REF = #next_motion.Data.SystemVariable.SysVarIdx
    DSVa:
      REF = #next_motion.Data.SystemVariable.AxIdx
    DSVd:
      REF = #next_motion.Data.SystemVariable.Data.R8_value
    DABNf:
      REF = #next_motion.Data.AutoBlockNumber.offset
    DABNo:
      REF = #next_motion.Data.AutoBlockNumber.factor
    DCSSPs:
      REF = #next_motion.Data.ConstantSurfaceSpeed.Speed
    DCSSPp:
      REF = #next_motion.Data.ConstantSurfaceSpeed.Programmed
    MXFPx:
      REF = #next_motion.Data.MXFrame.Pos.x
    MXFPy:
      REF = #next_motion.Data.MXFrame.Pos.y
    MXFPz:
      REF = #next_motion.Data.MXFrame.Pos.z
    MXFOt:
      REF = #next_motion.Data.MXFrame.Orient.Type
    MXFOa:
      REF = #next_motion.Data.MXFrame.Orient.Angle
    MXTFPx:
      REF = #next_motion.Data.MXTool.Frame.Pos.x
    MXTFPy:
      REF = #next_motion.Data.MXTool.Frame.Pos.y
    MXTFPz:
      REF = #next_motion.Data.MXTool.Frame.Pos.z
    MXTFOt:
      REF = #next_motion.Data.MXTool.Frame.Orient.Type
    MXTFOa:
      REF = #next_motion.Data.MXTool.Frame.Orient.Angle
    MXTr:
      REF = #next_motion.Data.MXTool.Radius
    MXPPx:
      REF = #next_motion.Data.MXPoint.Pos.x
    MXPPy:
      REF = #next_motion.Data.MXPoint.Pos.y
    MXPPz:
      REF = #next_motion.Data.MXPoint.Pos.z
    MXPOt:
      REF = #next_motion.Data.MXPoint.Orient.Type
    MXPOa:
      REF = #next_motion.Data.MXPoint.Orient.Angle
    MXPCm:
      REF = #next_motion.Data.MXPoint.Cfg.Mode
    MXPr:
      REF = #next_motion.Data.MXPoint.RotAxis
    MXPa:
      REF = #next_motion.Data.MXPoint.AuxAxis
    MXPhTr:
      REF = #next_motion.Data.MXPathDesc.Trans.Radius
    MXPhTt:
      REF = #next_motion.Data.MXPathDesc.Trans.Type
    MXDa:
      REF = #next_motion.Data.MXDynamicDesc.Accel
    MXDd:
      REF = #next_motion.Data.MXDynamicDesc.Decel
    MXDOe:
      REF = #next_motion.Data.MXDynamicDesc.Optmot.Enable
    MXDOv:
      REF = #next_motion.Data.MXDynamicDesc.Optmot.VelPathDef
    MXDOr:
      REF = #next_motion.Data.MXDynamicDesc.Optmot.RobotPar
    MXDOl:
      REF = #next_motion.Data.MXDynamicDesc.Optmot.Limits
    MXVv:
      REF = #next_motion.Data.MXVelocity.v
    MXVm:
      REF = #next_motion.Data.MXVelocity.Mode
    MXAj:
      REF = #next_motion.Data.MXAxisTarget.JointAxis
    MXAa:
      REF = #next_motion.Data.MXAxisTarget.AuxAxis
    MXAb:
      REF = #next_motion.Data.MXAxisTarget.BaseAxis
    MXJ:
      REF = #next_motion.Data.MXJointAxis
    MXAto:
      REF = #next_motion.Data.MXAutoTang.Offset
    MXCDCas:
      REF = #next_motion.Data.MXCDC.ArcTransSpd
    MXCDCsm:
      REF = #next_motion.Data.MXCDC.SpdMode
    MXCDCcv:
      REF = #next_motion.Data.MXCDC.ContourViolation
    MXCDCtm:
      REF = #next_motion.Data.MXCDC.TransMode
    MXCDCem:
      REF = #next_motion.Data.MXCDC.EntryMode
    MXCDCal:
      REF = #next_motion.Data.MXCDC.AcrToLine
    THCp:
      REF = #next_motion.Data.ThreadCut.Position
    THCi:
      SET = #next_motion.Data.ThreadCut.Idx[0] = ArrayRep(:(:-1:):);
        #next_motion.Data.ThreadCut.Idx = ${EXPR};
    THCm:
      SET = #next_motion.Data.ThreadCut.Mode[0] = ArrayRep(:(:-1:):);
        #next_motion.Data.ThreadCut.Mode = ${EXPR};
    THCld:
      REF = #next_motion.Data.ThreadCut.LeadDirection
    THCl:
      REF = #next_motion.Data.ThreadCut.Lead
    THCo:
      REF = #next_motion.Data.ThreadCut.Offset
    ACVc:
      REF = #next_motion.Data.AxisCtrlVelocity.Command
    ACVi:
      REF = #next_motion.Data.AxisCtrlVelocity.Idx
    ACSs:
      REF = #next_motion.Data.AxisCtrlSpeed.Speed
    ACSi:
      REF = #next_motion.Data.AxisCtrlSpeed.Idx
    ACPp:
      REF = #next_motion.Data.AxisCtrlPosition.Position
    ACPd:
      REF = #next_motion.Data.AxisCtrlPosition.PositionDefined
    ACPi:
      REF = #next_motion.Data.AxisCtrlPosition.Idx
    ACPm:
      REF = #next_motion.Data.AxisCtrlPosition.Mode
    CHFm:
      REF = #next_motion.Data.Champfer.Mode
    CHFv:
      REF = #next_motion.Data.Champfer.Value
    PAFv:
      REF = #next_motion.Data.PathFeed.Value
    PAFi:
      REF = #next_motion.Data.PathFeed.Id
    GENd:
      REF = #next_motion.Data.GenericData.Data
    SGALd:
      REF = #next_motion.Data.SetGmcAxisLimit.DestinationAxis
    SGALs:
      REF = #next_motion.Data.SetGmcAxisLimit.SourceAxis
    SGALn:
      SET = BlockCpy(:\#next_motion.Data.SetGmcAxisLimit.SourceLimitSetName, ${EXPR}:);
  Constants:
    PathBusy = BUSY (type=STRING)
    PathStatus = STATUS (type=STRING)
    PathErrLevel = ERRLEV (type=STRING)
  BuiltInProcs:
    SendCommand = SendCommand(:$[1]:); (MinArgs=1, MaxArgs=1, Inline=Yes)
    DispatchAndWait = DispatchAndWait(:$[1]:); (MinArgs=1, MaxArgs=1, Inline=Yes)
  Preprocess:
    MP_PJN (Search=MP22000 , Replace=PJN )
    MP_PJB (Search=MP22100 , Replace=PJB )
  GCodes:
    G_DELAY (GNum=0, Alias=@, AliasIsPattern=Yes, Inline=Yes)
      Arg (DataType=FLOAT, ref=tickdelay)
    G_PJN (GNum=22000, Alias=PJN, Inline=Yes, Group=220)
      Arg PathBusy (DataType=FLOAT, ref=busy_count)
      Arg PathStatus (DataType=FLOAT, ref=final_status)
      Arg PathErrLevel (DataType=FLOAT, ref=error_level)
    G_PJB (GNum=22100, Alias=PJB, Inline=Yes, Group=220)
      Arg PathBusy (DataType=FLOAT, ref=busy_count)
      Arg PathStatus (DataType=FLOAT, ref=final_status)
      Arg PathErrLevel (DataType=FLOAT, ref=error_level)
  MCodes:
    M_DEFAULT (IsDefault=Yes, MinValue=0, MaxValue=999999)
      ARG (ref=VALUE, DataType=FLOAT, RequireLiteral=Yes)
    M10003 = 10003 (Inline=Yes)
      ARG (ref=VALUE, DataType=FLOAT, RequireLiteral=Yes)
    M1000000 = 1000000 (Alias=;, AliasIsPattern=Yes, Inline=Yes, IgnoreIfGroups=220)
      ARG (ref=VALUE, DataType=FLOAT, RequireLiteral=Yes)
  ParserData (NestedComments=No, DefaultCaseSensitive=Yes, CommentsSpanLines=No, ReadWholeFileBeforeParsing=No, ExpectMainProgStmts=Yes, UseFubTemplates=No)
    TKG_END_OF_LINE = \n (IsPattern=No)
    TKG_OPEN_COMMENT = #
    TKG_NC_BLOCK_PREFIX = N:[\s\d] (IsPattern=Yes)
    TKG_OPEN_LISTBRACKET = (
    TKG_CLOSE_LISTBRACKET = )
    TKG_COMMA = ,
    TKG_NUMBER = \d+\.\d+|\d+\.|\.\d+ (IsPattern=Yes)
    TKG_INTEGER = \d+ (IsPattern=Yes)
    TKG_NUMBER_EXP = e:[\s\d\+\-\.] (IsPattern=Yes)
    TKG_ASSIGN_EQ = =
    TKG_ARITH_BINARY_MINUS = -
    TKG_M_CODE_PREFIX = MP:\d (IsPattern=Yes)
  StringChars (AsciiStringStart=")
    EscapeSeq (Search=$N, CaseSensitive=No, ReplaceValue=10)
    EscapeSeq (Search=$L, CaseSensitive=Yes, ReplaceValue=10)
    EscapeSeq (Search=$Q, CaseSensitive=No, ReplaceStr=")
    EscapeSeq (Search=$[\dA-F]+, IsPattern=Yes, CaseSensitive=No, ReplaceEncodingBase=16)
    EscapeSeq (Search=$$, ReplaceStr=$)
    EscapeSeq (Search=$, ReplaceStr=)
```

- Data object Logical/GmcIpConfig/gmcipesm (Cnc, version 3.13.0) (no source held here)

- Data object Logical/GmcIpConfig/gmcipmxd (Cnc, version 3.13.0) (no source held here)

### Data object Logical/GmcIpConfig/gmcipmx (Cnc)

#### gmcipmx.cnc
```
Root (LangModule=ailgcode, Version=1.0)
  AILHeader = sub OnProgStart
      %_Frm = %FRM_0;
      %_Base = %BASE_0;
      %_Tool = %TOOL_0;
      %_Vel = %VEL_0;
      %_Pth = %PTH_0;
      %_Dyn = %DYN_0;
      BlockCpy(:\%_Ref, \%REF_0:);
    endsub
  BuiltInProcs:
    WAIT_PP_SYNC = #next_motion.Command = MPCMD_IP_SYNCH_PP;
      PushPacket(::);
      DispatchAndWait(:IPCMD_SYNC_PP_CONT:);
    ERROR_EX = ErrorEx(:"id":$[1],"fmt":$[2],"data":(:$[3],$[4],$[5],$[6],$[7],$[8],$[9],$[10],$[11],$[12],$[13],$[14]:):); (MinArgs=3, MaxArgs=14)
    SET_POINT:
      Arg (ref=POINT, DataType=ANY_DATA, MinCount=1, MaxCount=1)
    SET_TRIGGER_CONFIG:
      Arg (ref=TRIGGER, DataType=ANY_DATA, MinCount=1, MaxCount=1)
      Arg (ref=bHALT, DataType=ANY_DATA, MinCount=1, MaxCount=1)
      Arg (ref=ID, DataType=ANY_DATA, MinCount=1, MaxCount=1)
    SET_WANTED_JOINT:
      Arg (ref=Ref, DataType=ANY_DATA, MinCount=1, MaxCount=1)
    SET_CIRCLE:
      Arg (ref=END_POINT, DataType=ANY_DATA, MinCount=1, MaxCount=1)
      Arg (ref=CIRCLE_POINT, DataType=ANY_DATA, MinCount=1, MaxCount=1)
      Arg (ref=Angle, DataType=IEC_LREAL, MinCount=0, MaxCount=1)
    SET_AXIS_TARGET:
      Arg (ref=AXIS_TARGET, DataType=ANY_DATA, MinCount=1, MaxCount=1)
    SET_FRAME:
      Arg (ref=Frm, DataType=ANY_DATA, MinCount=0, MaxCount=1)
    SET_BASEFRAME:
      Arg (ref=Base, DataType=ANY_DATA, MinCount=0, MaxCount=1)
    SET_TOOL:
      Arg (ref=Tool, DataType=ANY_DATA, MinCount=0, MaxCount=1)
    SET_PATH_DESC:
      Arg (ref=Pth, DataType=ANY_DATA, MinCount=0, MaxCount=1)
    SET_DYNAMIC_DESC:
      Arg (ref=Dyn, DataType=ANY_DATA, MinCount=0, MaxCount=1)
    SET_VELOCITY:
      Arg (ref=Vel, DataType=ANY_DATA, MinCount=0, MaxCount=1)
    JointToPoint:
      Arg (ref=Joint, UserType=MXJointAxisType, MinCount=1, MaxCount=1)
      Arg (ref=Point, UserType=MXPointType, MinCount=1, MaxCount=1)
    PointToJoint:
      Arg (ref=Point, UserType=MXPointType, MinCount=1, MaxCount=1)
      Arg (ref=Joint, UserType=MXJointAxisType, MinCount=1, MaxCount=1)
    MoveL:
      Arg (ref=POINT, UserType=MXPointType, MinCount=1, MaxCount=1)
      Arg (ref=Frm, UserType=MXFrameType, MinCount=0, MaxCount=1)
      Arg (ref=Base, UserType=MXFrameType, MinCount=0, MaxCount=1)
      Arg (ref=Tool, UserType=MXToolType, MinCount=0, MaxCount=1)
      Arg (ref=Vel, UserType=MXVelocityType, MinCount=0, MaxCount=1)
      Arg (ref=Pth, UserType=MXPathDescType, MinCount=0, MaxCount=1)
      Arg (ref=Dyn, UserType=MXDynamicDescType, MinCount=0, MaxCount=1)
    MoveJ:
      Arg (ref=POINT, UserType=MXPointType, MinCount=1, MaxCount=1)
      Arg (ref=Frm, UserType=MXFrameType, MinCount=0, MaxCount=1)
      Arg (ref=Base, UserType=MXFrameType, MinCount=0, MaxCount=1)
      Arg (ref=Tool, UserType=MXToolType, MinCount=0, MaxCount=1)
      Arg (ref=Vel, UserType=MXVelocityType, MinCount=0, MaxCount=1)
      Arg (ref=Ref, UserType=MXJointAxisType, MinCount=0, MaxCount=1)
      Arg (ref=Pth, UserType=MXPathDescType, MinCount=0, MaxCount=1)
      Arg (ref=Dyn, UserType=MXDynamicDescType, MinCount=0, MaxCount=1)
    MoveC:
      Arg (ref=END_POINT, UserType=MXPointType, MinCount=1, MaxCount=1)
      Arg (ref=CIRCLE_POINT, UserType=MXPointType, MinCount=1, MaxCount=1)
      Arg (ref=Angle, DataType=IEC_LREAL, MinCount=0, MaxCount=1)
      Arg (ref=Frm, UserType=MXFrameType, MinCount=0, MaxCount=1)
      Arg (ref=Base, UserType=MXFrameType, MinCount=0, MaxCount=1)
      Arg (ref=Tool, UserType=MXToolType, MinCount=0, MaxCount=1)
      Arg (ref=Vel, UserType=MXVelocityType, MinCount=0, MaxCount=1)
      Arg (ref=Pth, UserType=MXPathDescType, MinCount=0, MaxCount=1)
      Arg (ref=Dyn, UserType=MXDynamicDescType, MinCount=0, MaxCount=1)
    MoveA:
      Arg (ref=AXIS_TARGET, UserType=MXAxisTargetType, MinCount=1, MaxCount=1)
      Arg (ref=Vel, UserType=MXVelocityType, MinCount=0, MaxCount=1)
      Arg (ref=Dyn, UserType=MXDynamicDescType, MinCount=0, MaxCount=1)
      Arg (ref=Pth, UserType=MXPathDescType, MinCount=0, MaxCount=1)
    MoveLSearch:
      Arg (ref=POINT, UserType=MXPointType, MinCount=1, MaxCount=1)
      Arg (ref=TRIGGER, UserType=MXTriggerConfigType, MinCount=1, MaxCount=1)
      Arg (ref=bHALT, DataType=IEC_BOOL, MinCount=1, MaxCount=1)
      Arg (ref=ID, DataType=IEC_UINT, MinCount=1, MaxCount=1)
      Arg (ref=Frm, UserType=MXFrameType, MinCount=0, MaxCount=1)
      Arg (ref=Base, UserType=MXFrameType, MinCount=0, MaxCount=1)
      Arg (ref=Tool, UserType=MXToolType, MinCount=0, MaxCount=1)
      Arg (ref=Vel, UserType=MXVelocityType, MinCount=0, MaxCount=1)
      Arg (ref=Pth, UserType=MXPathDescType, MinCount=0, MaxCount=1)
      Arg (ref=Dyn, UserType=MXDynamicDescType, MinCount=0, MaxCount=1)
    WaitTime:
      Arg (ref=set_time, DataType=IEC_LREAL, MinCount=1, MaxCount=1)
    WaitIp = #next_motion.Command = MPCMD_IP_SYNCH;
      if (#restart.playback)
        #next_motion.Data.I4_value = ncSIMULATION;
      else
        #next_motion.Data.I4_value = ncSTANDARD;
      endif
      PushPacket(::);
      DispatchAndWait(:IPCMD_SYNC_PLC_CONT:);
    WaitEndMove = #next_motion.Command = MPCMD_IP_SYNCH_PATH;
      PushPacket(::);
      DispatchAndWait(:IPCMD_SYNC_PATH_CONT:);
    TmpTool = %__tmp_tool.Frame.Pos.x = %_CNC.tool_dx;
      %__tmp_tool.Frame.Pos.y = %_CNC.tool_dy;
      %__tmp_tool.Frame.Pos.z = %_CNC.tool_dz;
      %__tmp_tool.Frame.Orient.Type = %_CNC.tool_angles_type;
      %__tmp_tool.Frame.Orient.Angle[0] = %_CNC.tool_phi;
      %__tmp_tool.Frame.Orient.Angle[1] = %_CNC.tool_theta;
      %__tmp_tool.Frame.Orient.Angle[2] = %_CNC.tool_psi;
      %__tmp_tool.Frame.Orient.Angle[3] = 0;
      %__tmp_tool.Radius = #sys_vars.RAD;
    GetTool:
      Arg (ref=Tool, UserType=MXToolType, MinCount=1, MaxCount=1)
    TmpBaseFrame = %__tmp_frame.Pos.x = %_CNC.base_frame_dx;
      %__tmp_frame.Pos.y = %_CNC.base_frame_dy;
      %__tmp_frame.Pos.z = %_CNC.base_frame_dz;
      %__tmp_frame.Orient.Type = %_CNC.base_frame_angles_type;
      %__tmp_frame.Orient.Angle[0] = %_CNC.base_frame_phi;
      %__tmp_frame.Orient.Angle[1] = %_CNC.base_frame_theta;
      %__tmp_frame.Orient.Angle[2] = %_CNC.base_frame_psi;
      %__tmp_frame.Orient.Angle[3] = 0;
    GetBaseFrame:
      Arg (ref=Frame, UserType=MXFrameType, MinCount=1, MaxCount=1)
    GetJoint:
      Arg (ref=Joint, UserType=MXJointAxisType, MinCount=1, MaxCount=1)
    GetAxisTarget:
      Arg (ref=AxisTarget, UserType=MXAxisTargetType, MinCount=1, MaxCount=1)
    GetLatchPoint:
      Arg (ref=ID, DataType=IEC_UINT, MinCount=1, MaxCount=1)
      Arg (ref=Point, UserType=MXPointType, MinCount=1, MaxCount=1)
      Arg (ref=Event, DataType=IEC_BOOL, MinCount=1, MaxCount=1)
    GetPoint:
      Arg (ref=Point, UserType=MXPointType, MinCount=1, MaxCount=1)
    GetPointIntern = %__tmp_point = %POINT_0;
      
      local $i;
      $i=0;
      lbegin(1)
        %__tmp_axis_code[$i] = %_AX.axis_map[$i];
        %__tmp_axis_idx[$i] = %_AX.axis_map_idx[$i];
        $i = $i + 1;
      lend($i < GetIpInt(:300:))     
      %__mx_status =  MXCncAxesToPoint(:%_CNC.adr_trf_data_mx,  \%__tmp_set_pos, \%__tmp_point,   %_CNC.trf_type, %_CNC.angles_type, \%__tmp_axis_code, \%__tmp_axis_idx, GetIpInt(:300:) :);
      if (%__mx_status > 0)
        
        ErrorEx(:"id":10905,"fmt":"4d4d4d","data":(:GetCurLine(::),4,%__mx_status:):);
      endif
    CDCOn:
      Arg (ref=Direction, DataType=INT, MinCount=1, MaxCount=1)
      Arg (ref=CDC, UserType=MXCDCType, MinCount=0, MaxCount=1)
    CDCOff:
      Arg (ref=CDC, UserType=MXCDCType, MinCount=0, MaxCount=1)
    AutoTangOn:
      Arg (ref=Param, UserType=MXAutoTangType, MinCount=0, MaxCount=1)
    AutoTangOff = #next_motion.Command = MPCMD_MX_TANG_AX_OFF;
      PushPacket(::);
    SetM = local $i, $num_item;
      $i = 1;
      $num_item = ListLength(:${*}:);
      lbegin (1)
        #next_motion.Command = MPCMD_SET_M_FCT;
        #next_motion.Data.I4_value = ListItemValue(:${*}, $i:);  
        PushPacket(::);
        $i = $i + 1;
      lend($i <= $num_item)
      DispatchMPList(::); (MinArgs=1, MaxArgs=10)
  SysVars:
    TRF_DATA_MX $TRF_DATA_MX:
      GET = return %_CNC.adr_trf_data_mx; (ReturnType=IEC_UDINT)
```

### gmcipus.cnc
```
LANGS
```

- Data object Logical/GmcIpUserConfig/gmcipvar (Cnc, version 3.13.0) (no source held here)

### Program Logical/SDCAxisCtr (ANSIC)

#### Variables.var
```iecst
VAR
	min_task : INT := 7000;
	desired_speed : INT := 0;
	axis_X : FB_Axis;
	coil_powered : BOOL := FALSE;
	coil_pwm_value : {REDUND_UNREPLICABLE} INT := 200;
	fb_controller : FB_Controller;
	pwm_period : {REDUND_UNREPLICABLE} UINT := 200;
END_VAR
```

#### Main.c
```c
#include <bur/plctypes.h>

#ifdef _DEFAULT_INCLUDES
	#include <AsDefault.h>
#endif

void increase_counters(void);

void _INIT ProgramInit(void)
{
	//Устанваливаем типы SDC модулей
	AxisX_HW.EncIf1_Typ = ncSDC_ENC16;
	AxisX_HW.DiDoIf_Typ = ncSDC_DIDO;
	AxisX_HW.DrvIf_Typ = ncSDC_DRVSERVO16;

	//Устанавливаем имена переменных
	strcpy(AxisX_HW.EncIf1_Name, "AxisX_EncIf");
	strcpy(AxisX_HW.DrvIf_Name, "AxisX_DrvIf");
	strcpy(AxisX_HW.DiDoIf_Name, "AxisX_DiDoIf");

	//Устанавливаем входы готовности и нормальной работы
	AxisX_EncIf.iEncOK = 1;
	AxisX_DrvIf.iDrvOK = 1;
	AxisX_DrvIf.iStatusEnable = 1;
	AxisX_DiDoIf.iDriveReady = 1;

	fb_controller.dt = 0.002;
	fb_controller.k_i = 0.16;
	fb_controller.k_p = 0.0064;
	fb_controller.max_abs_value = 24.0;

	pwm_period = 200;
}

void _CYCLIC ProgramCyclic(void)
{
	FB_Axis(&axis_X);
	coil_pwm_value = coil_powered ? 32767 : 0;

	increase_counters();

	//Формирование показаний датчика

	AxisX_EncIf.iActTime = (INT)	AsIOTimeCyclicStart();
	AxisX_EncIf.iActPos = axis_X.counter;
	AxisX_DiDoIf.iPosHwEnd = axis_X.endswitch_a_reached;
	AxisX_DiDoIf.iNegHwEnd = axis_X.endswitch_b_reached;
	fb_controller.in = AxisX_DrvIf.oSetPos;

	if((fb_controller.in<min_task)&&(fb_controller.in>(-min_task))) fb_controller.in = 0;
	fb_controller.in = fb_controller.in * 6500/32767 - axis_X.speed;

	FB_Controller(&fb_controller);

	axis_X.pwm_value = fb_controller.out / 24.0 * 32767;
}

void increase_counters(void)
{
	AxisX_EncIf.iLifeCnt++;
	AxisX_DiDoIf.iLifeCntDriveEnable++;
	AxisX_DiDoIf.iLifeCntDriveReady++;
	AxisX_DiDoIf.iLifeCntNegHwEnd++;
	AxisX_DiDoIf.iLifeCntPosHwEnd++;
	AxisX_DiDoIf.iLifeCntReference++;
	AxisX_DrvIf.iLifeCnt++;
}

void _EXIT ProgramExit(void)
{
	// Insert code here

}
```

Listed in the project but not available here: Logical/Global.typ, Logical/AxisApt, Logical/Types.typ, Logical/AxisInit, Logical/acp10etxen, Logical/ncsdcctrl, Logical/GmcIpConfig/gmciplsm, Logical/GmcIpConfig/gmcipcfg, Logical/GmcIpConfig/gmcipiec, Logical/CncInit, Logical/CncProg
